Fanuc KAREL source: kc00030.KL

PROGRAM KC00030
%STACKSIZE=65535
%PRIORITY=65535
%NOLOCKGROUP
VAR
I : INTEGER
J : INTEGER
K : INTEGER
R : REAL
B : BOOLEAN
S : STRING[80]
T : STRING[80]
AI : ARRAY[8] OF INTEGER
BA : ARRAY[8] OF BOOLEAN
BC : ARRAY[8,8] OF BOOLEAN
SA : ARRAY[8] OF STRING[80]
VP : ARRAY[8,8] OF INTEGER
-- UNRESOLVED DECLARATIONS (source type spelling not recovered)
-- P : TYPE_0x001F (type_u16=0x001F)
-- Q : TYPE_0x001F (type_u16=0x001F)
-- AB : ARRAY[244] OF TYPE_0x0018 (type_u16=0x2018)
-- CD : ARRAY[8] OF TYPE_0x1102 (type_u16=0x3102)
-- X : TYPE_0x1103 (type_u16=0x1103)
BEGIN
S='DICT'
INIT_TBL(S,I,J,K,CD,BA,BC,SA,VP,X,I)
END KC00030
